INTERFACE I_Layer EXTENDS I_Component

{attribute 'OPC.UA.DA.Property' := '1'}
{attribute 'monitoring' := 'call'}
PROPERTY P_List : I_ListComponent
GET
END_GET
END_PROPERTY

METHOD PUBLIC M_Attach
VAR_INPUT
	iComponent:		I_Component;
END_VAR
END_METHOD

METHOD PUBLIC M_Dettach
VAR_INPUT
	iComponent:		I_Component;
END_VAR
END_METHOD

{attribute 'OPC.UA.DA.Property' := '1'}
{attribute 'monitoring' := 'call'}
PROPERTY PUBLIC P_Next : I_Component
GET
END_GET
SET
END_SET
END_PROPERTY

END_INTERFACE

(* stored: Version 1.1.0.1
   Itf I_Layer: Id {8f4734e9-8603-08d1-26cb-b0fac42f0340}
   Property P_List: Id {5f16ca22-2e9f-0624-17c9-8649b64dfee2}
   Get Get: Id {02a31d1a-c1c4-0420-3d69-4899685629b3}
   Method M_Attach: Id {79642475-2d99-0bbf-2634-5569c28ece9f}
   Method M_Dettach: Id {c474b0cc-3eba-08ca-0ece-5ec0960fd264}
   Property P_Next: Id {e45d8bd2-ecda-0a90-05dc-dc02c54ffcca}
   Get Get: Id {02e4ba9f-3195-05b1-1565-7ea4f5d3924f}
   Set Set: Id {ddb2951c-a0b5-041c-2026-704c21188550} *)
